(* IEC 61131-3 sources: tutorials/projects/ch08-1/PROGRAM, 2 files *)

(* ---- MC_Auto_Gen.ST ---- *)
(* This is automatically generated file, don't modify it *)

CONFIGURATION axis_config
    VAR_GLOBAL
        Axis1: AXIS_REF;
    END_VAR
END_CONFIGURATION

FUNCTION MC_Init_Axis
    VAR_EXTERNAL
        Axis1: AXIS_REF;
    END_VAR

    Axis1 := mc_axis_create('Axis1');
    mc_axis_assign_servo(Axis1, mc_servo_new_DS402());

END_FUNCTION

(* ---- prog_main.st ---- *)
PROGRAM PLC_PRG
    VAR
        fbPower: MC_Power; (* 定义功能块实例 *)
        fbHome: MC_Home;
        fbMoveVel: MC_MoveVelocity;
        fbStop: MC_Stop;
        power_valid: BOOL;
    END_VAR

    fbPower(Axis := Axis1, Enable := TRUE, EnablePositive := TRUE, EnableNegative := TRUE, Valid => power_valid);
    IF NOT fbPower.Status THEN
       RETURN;
    END_IF;

    fbHome(Axis := Axis1, Execute := TRUE, Position := 0, BufferMode := 0 /*mcAborting*/);

    fbMoveVel(Axis := Axis1, Execute := fbHome.Done, ContinuousUpdate:= TRUE, Velocity:=100);

    fbStop(Axis := Axis1, Execute := fbMoveVel.InVelocity);

END_PROGRAM
